FUNCTION_BLOCK TestFB
VAR_INPUT
END_VAR
VAR_OUTPUT
END_VAR
VAR
END_VAR

// NETWORK 1

END_FUNCTION_BLOCK

(* stored: Version 1.1.0.1, ProductVersion 3.1.4024.10
   POU TestFB: Id {e9d99044-0a14-4650-af41-1fe80cc14c6b}, SpecialFunc None *)
